PROGRAM MAIN1
VAR
	counter1, edge, FALL     :UDINT;
	COUNTONESECPULSE: BLINK;
	sw1 : BOOL;
	COUNTER2: INT;
	posedge : R_TRIG;
	negedge: F_TRIG;
	SW3: BOOL;
END_VAR


counter1 := counter1 +1 ;


COUNTONESECPULSE(ENABLE:= GVL.S3, TIMELOW:= T#500MS , TIMEHIGH:=T#500MS , OUT=> GVL.flasher );


	posedge(CLK:=GVL.flasher , Q=> );
	
	edge := edge + TO_UDINT(posedge.Q);
	
	negedge(CLK:=GVL.flasher , Q=> );
	
	fall := fall + TO_UDINT(negedge.Q);
	
	GVL.LED4 		:= FALSE;
	
	
IF GVL.S4 THEN
	GVL.LED4		:= TRUE;
	edge			 := 0;
	fall			 :=0 ;
	counter1 		 := 0;
	GVL.counter      :=0;
	GVL.flasher		 := fALSE;
END_IF

END_PROGRAM

(* stored: Version 1.1.0.1, ProductVersion 3.1.4024.12
   POU MAIN1: Id {b87cb413-83c0-40ae-b8e8-1063006edf74}, SpecialFunc None *)
